FUNCTION_BLOCK Serializer4Way
  (* Version 1.0, 2005-11-21, Goran Cengic, Chalmers *)
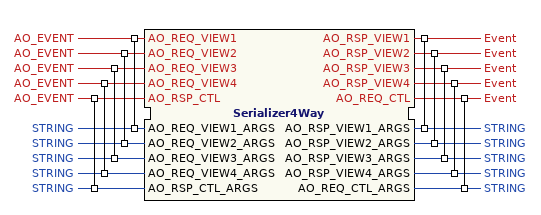
  EVENT_INPUT
    AO_REQ_VIEW1 : AO_EVENT WITH AO_REQ_VIEW1_ARGS;
    AO_REQ_VIEW2 : AO_EVENT WITH AO_REQ_VIEW2_ARGS;
    AO_REQ_VIEW3 : AO_EVENT WITH AO_REQ_VIEW3_ARGS;
    AO_REQ_VIEW4 : AO_EVENT WITH AO_REQ_VIEW4_ARGS;
    AO_RSP_CTL : AO_EVENT WITH AO_RSP_CTL_ARGS;
  END_EVENT
  EVENT_OUTPUT
    AO_RSP_VIEW1 WITH AO_RSP_VIEW1_ARGS;
    AO_RSP_VIEW2 WITH AO_RSP_VIEW2_ARGS;
    AO_RSP_VIEW3 WITH AO_RSP_VIEW3_ARGS;
    AO_RSP_VIEW4 WITH AO_RSP_VIEW4_ARGS;
    AO_REQ_CTL WITH AO_REQ_CTL_ARGS;
  END_EVENT
  VAR_INPUT
    AO_REQ_VIEW1_ARGS : STRING;
    AO_REQ_VIEW2_ARGS : STRING;
    AO_REQ_VIEW3_ARGS : STRING;
    AO_REQ_VIEW4_ARGS : STRING;
    AO_RSP_CTL_ARGS : STRING;
  END_VAR
  VAR_OUTPUT
    AO_RSP_VIEW1_ARGS : STRING;
    AO_RSP_VIEW2_ARGS : STRING;
    AO_RSP_VIEW3_ARGS : STRING;
    AO_RSP_VIEW4_ARGS : STRING;
    AO_REQ_CTL_ARGS : STRING;
  END_VAR
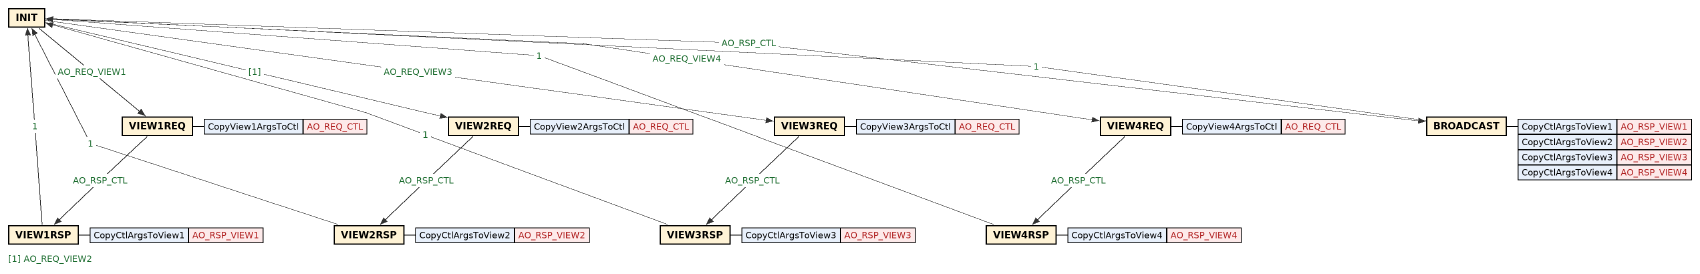
  EC_STATES
    INIT;
    VIEW1REQ : CopyView1ArgsToCtl -> AO_REQ_CTL;
    VIEW1RSP : CopyCtlArgsToView1 -> AO_RSP_VIEW1;
    INIT;
    VIEW2REQ : CopyView2ArgsToCtl -> AO_REQ_CTL;
    VIEW2RSP : CopyCtlArgsToView2 -> AO_RSP_VIEW2;
    INIT;
    VIEW3REQ : CopyView3ArgsToCtl -> AO_REQ_CTL;
    VIEW3RSP : CopyCtlArgsToView3 -> AO_RSP_VIEW3;
    INIT;
    VIEW4REQ : CopyView4ArgsToCtl -> AO_REQ_CTL;
    VIEW4RSP : CopyCtlArgsToView4 -> AO_RSP_VIEW4;
    INIT;
    BROADCAST : CopyCtlArgsToView1 -> AO_RSP_VIEW1, CopyCtlArgsToView2 -> AO_RSP_VIEW2, CopyCtlArgsToView3 -> AO_RSP_VIEW3, CopyCtlArgsToView4 -> AO_RSP_VIEW4;
  END_STATES
  EC_TRANSITIONS
    INIT TO VIEW1REQ := AO_REQ_VIEW1;
    VIEW1REQ TO VIEW1RSP := AO_RSP_CTL;
    VIEW1RSP TO INIT := 1;
    INIT TO VIEW2REQ := AO_REQ_VIEW2;
    VIEW2REQ TO VIEW2RSP := AO_RSP_CTL;
    VIEW2RSP TO INIT := 1;
    INIT TO VIEW3REQ := AO_REQ_VIEW3;
    VIEW3REQ TO VIEW3RSP := AO_RSP_CTL;
    VIEW3RSP TO INIT := 1;
    INIT TO VIEW4REQ := AO_REQ_VIEW4;
    VIEW4REQ TO VIEW4RSP := AO_RSP_CTL;
    VIEW4RSP TO INIT := 1;
    INIT TO BROADCAST := AO_RSP_CTL;
    BROADCAST TO INIT := 1;
  END_TRANSITIONS
  ALGORITHM CopyView1ArgsToCtl IN Java:
	    AO_REQ_CTL_ARGS = AO_REQ_VIEW1_ARGS;
  END_ALGORITHM
  ALGORITHM CopyCtlArgsToView1 IN Java:
	    AO_RSP_VIEW1_ARGS = AO_RSP_CTL_ARGS;
  END_ALGORITHM
  ALGORITHM CopyView2ArgsToCtl IN Java:
	    AO_REQ_CTL_ARGS = AO_REQ_VIEW2_ARGS;
  END_ALGORITHM
  ALGORITHM CopyCtlArgsToView2 IN Java:
	    AO_RSP_VIEW2_ARGS = AO_RSP_CTL_ARGS;
  END_ALGORITHM
  ALGORITHM CopyView3ArgsToCtl IN Java:
	    AO_REQ_CTL_ARGS = AO_REQ_VIEW3_ARGS;
  END_ALGORITHM
  ALGORITHM CopyCtlArgsToView3 IN Java:
	    AO_RSP_VIEW3_ARGS = AO_RSP_CTL_ARGS;
  END_ALGORITHM
  ALGORITHM CopyView4ArgsToCtl IN Java:
	    AO_REQ_CTL_ARGS = AO_REQ_VIEW4_ARGS;
  END_ALGORITHM
  ALGORITHM CopyCtlArgsToView4 IN Java:
	    AO_RSP_VIEW4_ARGS = AO_RSP_CTL_ARGS;
  END_ALGORITHM
END_FUNCTION_BLOCK
(* other elements stored in the file *)
(* View 1 *)
(* View 2 *)
(* View 3 *)
(* View 4 *)
(* Broadcast to all views *)
